ABB RAPID module: A057_DataTask_1.mod

MODULE A057_DataTask_1
    !***********************************************************************************
    !
    ! ETH Zurich / NCCR Digital Fabrication
    ! HIB C51 / Stefano-Franscini-Platz 1
    ! CH-8093 Zürich
    !
    !***********************************************************************************
    !
    ! PROJECT     :  A057 MAS Rio
    !
    ! FUNCTION    :  Includ all Task Data's for Project
    !
    ! AUTHOR      :  Philippe Fleischmann
    !
    ! EMAIL       :  fleischmann@arch.ethz.ch
    !
    ! HISTORY     :  2020.01.27
    !
    ! Copyright   :  ETH Zürich (CH) 2019
    !
    !***********************************************************************************

    !************************************************
    ! Declaration :     bool
    !************************************************
    !

    !************************************************
    ! Declaration :     num
    !************************************************
    !

    !************************************************
    ! Declaration :     string
    !************************************************
    !

    !************************************************
    ! Declaration :     tooldata
    !************************************************
    !
    TASK PERS tooldata t_A057_ClayTool02:=[TRUE,[[0,0,354],[1,0,0,0]],[5,[10,0,55],[1,0,0,0],0,0,0]];

    TASK PERS tooldata t_A057_ClayTool02_Prism:=[TRUE,[[111.624,17.600,189.561],[1,0,0,0]],[5.0,[0.0,0.0,100],[1,0,0,0],0,0,0]];
    !TASK PERS tooldata t_A057_ClayTool02_DistSensor:=[TRUE,[[-113.660,-18.776,212.410],[1,0,0,0]],[1.000,[0.000,0.000,100.000],[1,0,0,0],0,0,0]];

    TASK PERS tooldata t_A057_ClayTool02_RealSense:=[TRUE,[[-149.558,-9.30087,234.713],[0.707106781,0,0,0.707106781]],[5,[0,0,100],[1,0,0,0],0,0,0]];
    TASK PERS tooldata t_A057_CalibrationNeedle:=[TRUE,[[0.693793,0.259468,245.505],[1,0,0,0]],[2,[0,0,50],[1,0,0,0],0,0,0]];

    !************************************************
    ! Declaration :     wobjdata
    !************************************************
    !
    TASK PERS wobjdata ob_A057_WobjPicking01:=[FALSE,TRUE,"",[[465.984,-1228.32,-46.0527],[0.00401767,-0.00103673,-0.00119599,-0.999991]],[[0,0,0],[1,0,0,0]]];
    TASK PERS wobjdata ob_A057_WobjPlacing01:=[FALSE,TRUE,"",[[359.262,2160.38,0],[1,0,0,0]],[[0,0,0],[1,0,0,0]]];

    !************************************************
    ! Declaration :     jointtarget
    !************************************************
    !
    TASK PERS jointtarget jp_A057_Jointtarget:=[[0,0,0,0,0,0],[9E9,9E9,9E9,9E9,9E9,9E9]];

    !************************************************
    ! Declaration :     robtarget
    !************************************************
    !
    TASK PERS robtarget p_A057_Robtarget:=[[0,0,0],[1,0,0,0],[0,0,0,0],[9E9,9E9,9E9,9E9,9E9,9E9]];

    !************************************************
    ! Declaration :     speeddata
    !************************************************
    !
    TASK PERS speeddata v_A057_Speed:=[0,0,0,0];
    TASK PERS tooldata t_A057_ClayTool_Mushroom:=[TRUE,[[0,0,105],[1,0,0,0]],[5,[10,0,55],[1,0,0,0],0,0,0]];
    TASK PERS tooldata t_A057_ClayTool_Egyptian:=[TRUE,[[-336.992,37.7122,44.7221],[0,0,1,0]],[5,[10,0,55],[1,0,0,0],0,0,0]];

ENDMODULE
